ABB RAPID module: CommonData.mod

MODULE CommonData

    ! Shared robtargets
    PERS robtarget pHome;
    PERS robtarget pStart;

ENDMODULE
